(* IEC 61131-3 sources: julia_exos_development/src/StringAndArray/StringAndA_0, 2 files *)

(* ---- StringAndArray.st ---- *)
PROGRAM _INIT

    StringAndArrayInit_0();

END_PROGRAM

PROGRAM _CYCLIC

    //Auto connect:
    //StringAndArrayCyclic_0.Enable := ExComponentInfo_0.Operational; // Component has been deployed and started up successfully

    StringAndArrayCyclic_0(Handle := StringAndArrayInit_0.Handle, pStringAndArray := ADR(StringAndArray_0));

    ExComponentInfo_0(ExTargetLink := ADR(gTarget_0), ExComponentLink := ADR(gStringAndArray_0), Enable := TRUE);

    ExDatamodelInfo_0(ExTargetLink := ADR(gTarget_0), Enable := TRUE, InstanceName := 'StringAndArray_0');

END_PROGRAM

PROGRAM _EXIT

    StringAndArrayExit_0(Handle := StringAndArrayInit_0.Handle);

END_PROGRAM

(* ---- StringAndArray.var ---- *)
VAR
    StringAndArrayInit_0 : StringAndArrayInit;
    StringAndArrayCyclic_0 : StringAndArrayCyclic;
    StringAndArrayExit_0 : StringAndArrayExit;
    StringAndArray_0 : StringAndArray;
    ExComponentInfo_0 : ExComponentInfo;
    ExDatamodelInfo_0 : ExDatamodelInfo;
END_VAR
